// TIA Portal V18 export
VAR_GLOBAL   // PLC tag table "Default tag table"
   "AI11.02.01" AT %IW96 : Int;
   "AI12.01.01" AT %IW68 : Int;
   "AI12.01.02" AT %IW70 : Int;
   "AI12.01.03" AT %IW72 : Int;
   "AI12.01.04" AT %IW74 : Int;
   "AI12.01.05" AT %IW76 : Int;
   "AI12.01.06" AT %IW78 : Int;
   "AI12.01.07" AT %IW80 : Int;
   "AI12.01.08" AT %IW82 : Int;
   "AI11.02.02" AT %IW98 : Int;
   "AI11.02.03" AT %IW100 : Int;
   "AI11.02.04" AT %IW102 : Int;
   "AI11.02.05" AT %IW104 : Int;
   "AI11.02.06" AT %IW106 : Int;
   "AI11.02.07" AT %IW108 : Int;
   "AI11.02.08" AT %IW110 : Int;
   "AI11.03.01" AT %IW112 : Int;
   "AI11.03.02" AT %IW114 : Int;
   "AI11.03.03" AT %IW116 : Int;
   "AI11.03.04" AT %IW118 : Int;
   "AI11.03.05" AT %IW120 : Int;
   "AI11.03.06" AT %IW122 : Int;
   "AI11.03.07" AT %IW124 : Int;
   "AI11.03.08" AT %IW126 : Int;
   "AO12.02.01" AT %QW68 : Int;
   "AO12.02.02" AT %QW70 : Int;
   "AO12.02.03" AT %QW72 : Int;
   "AO12.02.04" AT %QW74 : Int;
   "AO12.02.05" AT %QW76 : Int;
   "AO12.02.06" AT %QW78 : Int;
   "AO12.02.07" AT %QW80 : Int;
   "AO12.02.08" AT %QW82 : Int;
   "DI12.03.01" AT %I2.0 : Bool;
   "DI12.03.02" AT %I2.1 : Bool;
   "DI12.03.03" AT %I2.2 : Bool;
   "DI12.03.04" AT %I2.3 : Bool;
   "DI12.03.05" AT %I2.4 : Bool;
   "DI12.03.06" AT %I2.5 : Bool;
   "DI12.03.07" AT %I2.6 : Bool;
   "DI12.03.08" AT %I2.7 : Bool;
   "DI12.03.09" AT %I3.0 : Bool;
   "DI12.03.10" AT %I3.1 : Bool;
   "DI12.03.11" AT %I3.2 : Bool;
   "DI12.03.12" AT %I3.3 : Bool;
   "DI12.03.13" AT %I3.4 : Bool;
   "DI12.03.14" AT %I3.5 : Bool;
   "DI12.03.15" AT %I3.6 : Bool;
   "DI12.03.16" AT %I3.7 : Bool;
   "DI12.03.17" AT %I4.0 : Bool;
   "DI12.03.18" AT %I4.1 : Bool;
   "DI12.03.19" AT %I4.2 : Bool;
   "DI12.03.20" AT %I4.3 : Bool;
   "DI12.03.21" AT %I4.4 : Bool;
   "DI12.03.22" AT %I4.5 : Bool;
   "DI12.03.23" AT %I4.6 : Bool;
   "DI12.03.24" AT %I4.7 : Bool;
   "DI12.03.25" AT %I5.0 : Bool;
   "DI12.03.26" AT %I5.1 : Bool;
   "DI12.03.27" AT %I5.2 : Bool;
   "DI12.03.28" AT %I5.3 : Bool;
   "DI12.03.29" AT %I5.4 : Bool;
   "DI12.03.30" AT %I5.5 : Bool;
   "DI12.03.31" AT %I5.6 : Bool;
   "DI12.03.32" AT %I5.7 : Bool;
   "DO12.04.01" AT %Q2.0 : Bool;
   "DO12.04.02" AT %Q2.1 : Bool;
   "DO12.04.03" AT %Q2.2 : Bool;
   "DO12.04.04" AT %Q2.3 : Bool;
   "DO12.04.05" AT %Q2.4 : Bool;
   "DO12.04.06" AT %Q2.5 : Bool;
   "DO12.04.07" AT %Q2.6 : Bool;
   "DO12.04.08" AT %Q2.7 : Bool;
   "DO12.04.09" AT %Q3.0 : Bool;
   "DO12.04.10" AT %Q3.1 : Bool;
   "DO12.04.11" AT %Q3.2 : Bool;
   "DO12.04.12" AT %Q3.3 : Bool;
   "DO12.04.13" AT %Q3.4 : Bool;
   "DO12.04.14" AT %Q3.5 : Bool;
   "DO12.04.15" AT %Q3.6 : Bool;
   "DO12.04.16" AT %Q3.7 : Bool;
   "DO12.04.17" AT %Q4.0 : Bool;
   "DO12.04.18" AT %Q4.1 : Bool;
   "DO12.04.19" AT %Q4.2 : Bool;
   "DO12.04.20" AT %Q4.3 : Bool;
   "DO12.04.21" AT %Q4.4 : Bool;
   "DO12.04.22" AT %Q4.5 : Bool;
   "DO12.04.23" AT %Q4.6 : Bool;
   "DO12.04.24" AT %Q4.7 : Bool;
   "DO12.04.25" AT %Q5.0 : Bool;
   "DO12.04.26" AT %Q5.1 : Bool;
   "DO12.04.27" AT %Q5.2 : Bool;
   "DO12.04.28" AT %Q5.3 : Bool;
   "DO12.04.29" AT %Q5.4 : Bool;
   "DO12.04.30" AT %Q5.5 : Bool;
   "DO12.04.31" AT %Q5.6 : Bool;
   "DO12.04.32" AT %Q5.7 : Bool;
   "DI11.05.01" AT %I16.0 : Bool;
   "DI11.05.02" AT %I16.1 : Bool;
   "DI11.05.03" AT %I16.2 : Bool;
   "DI11.05.04" AT %I16.3 : Bool;
   "DI11.05.05" AT %I16.4 : Bool;
   "DI11.05.06" AT %I16.5 : Bool;
   "DI11.05.07" AT %I16.6 : Bool;
   "DI11.05.08" AT %I16.7 : Bool;
   "DI11.05.09" AT %I17.0 : Bool;
   "DI11.05.10" AT %I17.1 : Bool;
   "DI11.05.11" AT %I17.2 : Bool;
   "DI11.05.12" AT %I17.3 : Bool;
   "DI11.05.13" AT %I17.4 : Bool;
   "DI11.05.14" AT %I17.5 : Bool;
   "DI11.05.15" AT %I17.6 : Bool;
   "DI11.05.16" AT %I17.7 : Bool;
   "DI11.06.01" AT %I20.0 : Bool;
   "DI11.06.02" AT %I20.1 : Bool;
   "DI11.06.03" AT %I20.2 : Bool;
   "DI11.06.04" AT %I20.3 : Bool;
   "DI11.06.05" AT %I20.4 : Bool;
   "DI11.06.06" AT %I20.5 : Bool;
   "DI11.06.07" AT %I20.6 : Bool;
   "DI11.06.08" AT %I20.7 : Bool;
   "DI11.06.09" AT %I21.0 : Bool;
   "DI11.06.10" AT %I21.1 : Bool;
   "DI11.06.11" AT %I21.2 : Bool;
   "DI11.06.12" AT %I21.3 : Bool;
   "DI11.06.13" AT %I21.4 : Bool;
   "DI11.06.14" AT %I21.5 : Bool;
   "DI11.06.15" AT %I21.6 : Bool;
   "DI11.06.16" AT %I21.7 : Bool;
   "DI11.07.01" AT %I28.0 : Bool;
   "DI11.07.02" AT %I28.1 : Bool;
   "DI11.07.03" AT %I28.2 : Bool;
   "DI11.07.04" AT %I28.3 : Bool;
   "DI11.07.05" AT %I28.4 : Bool;
   "DI11.07.06" AT %I28.5 : Bool;
   "DI11.07.07" AT %I28.6 : Bool;
   "DI11.07.08" AT %I28.7 : Bool;
   "DI11.07.09" AT %I29.0 : Bool;
   "DI11.07.10" AT %I29.1 : Bool;
   "DI11.07.11" AT %I29.2 : Bool;
   "DI11.07.12" AT %I29.3 : Bool;
   "DI11.07.13" AT %I29.4 : Bool;
   "DI11.07.14" AT %I29.5 : Bool;
   "DI11.07.15" AT %I29.6 : Bool;
   "DI11.07.16" AT %I29.7 : Bool;
   "DO11.07.01" AT %Q28.0 : Bool;
   "DO11.07.02" AT %Q28.1 : Bool;
   "DO11.07.03" AT %Q28.2 : Bool;
   "DO11.07.04" AT %Q28.3 : Bool;
   "DO11.07.05" AT %Q28.4 : Bool;
   "DO11.07.06" AT %Q28.5 : Bool;
   "DO11.07.07" AT %Q28.6 : Bool;
   "DO11.07.08" AT %Q28.7 : Bool;
   "DO11.07.09" AT %Q29.0 : Bool;
   "DO11.07.10" AT %Q29.1 : Bool;
   "DI11.08.01" AT %I32.0 : Bool;
   "DI11.08.02" AT %I32.1 : Bool;
   "DI11.08.03" AT %I32.2 : Bool;
   "DI11.08.04" AT %I32.3 : Bool;
   "DI11.08.05" AT %I32.4 : Bool;
   "DI11.08.06" AT %I32.5 : Bool;
   "DI11.08.07" AT %I32.6 : Bool;
   "DI11.08.08" AT %I32.7 : Bool;
   "DI11.08.09" AT %I33.0 : Bool;
   "DI11.08.10" AT %I33.1 : Bool;
   "DI11.08.11" AT %I33.2 : Bool;
   "DI11.08.12" AT %I33.3 : Bool;
   "DI11.08.13" AT %I33.4 : Bool;
   "DI11.08.14" AT %I33.5 : Bool;
   "DI11.08.15" AT %I33.6 : Bool;
   "DI11.08.16" AT %I33.7 : Bool;
   "DI11.01.01" AT %I0.0 : Bool;
   "DI11.01.02" AT %I0.1 : Bool;
   "DI11.01.03" AT %I0.2 : Bool;
   "DI11.01.04" AT %I0.3 : Bool;
   "DI11.01.05" AT %I0.4 : Bool;
   "DI11.01.06" AT %I0.5 : Bool;
   "DI11.01.07" AT %I0.6 : Bool;
   "DI11.01.08" AT %I0.7 : Bool;
   "DI11.01.09" AT %I1.0 : Bool;
   "DI11.01.10" AT %I1.1 : Bool;
   "DI11.01.11" AT %I1.2 : Bool;
   "DI11.01.12" AT %I1.3 : Bool;
   "DI11.01.13" AT %I1.4 : Bool;
   "DI11.01.14" AT %I1.5 : Bool;
   "DO11.07.11" AT %Q29.2 : Bool;
   "DO11.07.12" AT %Q29.3 : Bool;
   "DO11.07.13" AT %Q29.4 : Bool;
   "DO11.07.14" AT %Q29.5 : Bool;
   "DO11.07.15" AT %Q29.6 : Bool;
   "DO11.07.16" AT %Q29.7 : Bool;
   "DO11.08.01" AT %Q32.0 : Bool;
   "DO11.08.02" AT %Q32.1 : Bool;
   "DO11.08.03" AT %Q32.2 : Bool;
   "DO11.08.04" AT %Q32.3 : Bool;
   "DO11.08.05" AT %Q32.4 : Bool;
   "DO11.08.06" AT %Q32.5 : Bool;
   "DO11.08.07" AT %Q32.6 : Bool;
   "DO11.08.08" AT %Q32.7 : Bool;
   "DO11.08.09" AT %Q33.0 : Bool;
   "DO11.08.10" AT %Q33.1 : Bool;
   "DO11.08.11" AT %Q33.2 : Bool;
   "DO11.08.12" AT %Q33.3 : Bool;
   "DO11.08.13" AT %Q33.4 : Bool;
   "DO11.08.14" AT %Q33.5 : Bool;
   "DO11.08.15" AT %Q33.6 : Bool;
   "DO11.08.16" AT %Q33.7 : Bool;
   "AO11.04.01" AT %QW128 : Int;
   "AO11.04.02" AT %QW130 : Int;
   "AO11.04.03" AT %QW132 : Int;
   "AO11.04.04" AT %QW134 : Int;
   "DO11.01.01" AT %Q0.0 : Bool;
   "DO11.01.02" AT %Q0.1 : Bool;
   "DO11.01.03" AT %Q0.2 : Bool;
   "DO11.01.04" AT %Q0.3 : Bool;
   "DO11.01.05" AT %Q0.4 : Bool;
   "DO11.01.06" AT %Q0.5 : Bool;
   "DO11.01.07" AT %Q0.6 : Bool;
   "DO11.01.08" AT %Q0.7 : Bool;
   "DO11.01.09" AT %Q1.0 : Bool;
   "DO11.01.10" AT %Q1.1 : Bool;
   "AI11.01.01" AT %IW64 : Int;
   "AI11.01.02" AT %IW66 : Int;
   "AO11.01.01" AT %QW64 : Int;
   "AO11.01.02" AT %QW66 : Int;
   System_Byte AT %MB1 : Byte;
   FirstScan AT %M1.0 : Bool;
   DiagStatusUpdate AT %M1.1 : Bool;
   AlwaysTRUE AT %M1.2 : Bool;
   AlwaysFALSE AT %M1.3 : Bool;
   Clock_Byte AT %MB0 : Byte;
   Clock_10Hz AT %M0.0 : Bool;
   Clock_5Hz AT %M0.1 : Bool;
   "Clock_2.5Hz" AT %M0.2 : Bool;
   Clock_2Hz AT %M0.3 : Bool;
   "Clock_1.25Hz" AT %M0.4 : Bool;
   Clock_1Hz AT %M0.5 : Bool;
   "Clock_0.625Hz" AT %M0.6 : Bool;
   "Clock_0.5Hz" AT %M0.7 : Bool;
   Lux AT %MD20 : Real;
   "DI12.05.01" AT %I6.0 : Bool;
   "DI12.05.02" AT %I6.1 : Bool;
   "DI12.05.03" AT %I6.2 : Bool;
   "DI12.05.04" AT %I6.3 : Bool;
   "DI12.05.05" AT %I6.4 : Bool;
   "DI12.05.06" AT %I6.5 : Bool;
   "DI12.05.07" AT %I6.6 : Bool;
   "DI12.05.08" AT %I6.7 : Bool;
   "DI12.05.09" AT %I7.0 : Bool;
   "DI12.05.10" AT %I7.1 : Bool;
   "DI12.05.11" AT %I7.2 : Bool;
   "DI12.05.12" AT %I7.3 : Bool;
   "DI12.05.13" AT %I7.4 : Bool;
   "DI12.05.14" AT %I7.5 : Bool;
   "DI12.05.15" AT %I7.6 : Bool;
   "DI12.05.16" AT %I7.7 : Bool;
   OAT_clock_triger AT %M5.0 : Bool;
   "Run/Stop" AT %M5.1 : Bool;
   rAO_temporary AT %MD60 : Real;
   rAI_temporary AT %MD61 : Real;
   xDO_temporary AT %M5.2 : Bool;   //    {ExternalWritable false}
   xDI_temporary AT %M5.3 : Bool;
   iUnitStateCounter AT %MW66 : Int;
   iTargetUnitStareCounter AT %MW68 : Int;
   cTargetUnitStatePrevOne AT %MB8 : Byte;
   cActualOpModePrevOne AT %MB9 : Byte;
   iActualOpModeCounter AT %MW10 : Int;
   xDL_Pump1_Run AT %M12.0 : Bool;
   xDL_Pump2_Run AT %M12.1 : Bool;
END_VAR
VAR_GLOBAL CONSTANT   // user constants
   IOmark_string_length : Int := 25;
   DIbasic_OnDelayCycle : Int := 800;
   DIbasic_OffDelayCycle : Int := 800;
END_VAR
